// normalize the input vector
FUNCTION vecNorm : LREAL
VAR_IN_OUT CONSTANT
	vec :ARRAY[*] OF LREAL;
END_VAR
VAR
	m,i:DINT;
END_VAR

m:=UPPER_BOUND(vec,1);
vecNorm:=0;
FOR i:=1 TO m DO
	vecNorm := vecNorm + vec[i]*vec[i];
END_FOR

END_FUNCTION

(* stored: Version 1.1.0.1, ProductVersion 3.1.4024.12
   POU vecNorm: Id {0015b5c6-4029-411f-8387-131591190194}, SpecialFunc None *)
